// TwinCAT 3 PLC project Main
// ProgramVersion: 3.1.4024.0
// libraries:
//   Tc2_Standard, * (Beckhoff Automation GmbH)
//   Tc2_System, * (Beckhoff Automation GmbH)
//   Tc3_Module, * (Beckhoff Automation GmbH)
//   VisuDialogs, * (System)
//   VisuSymbols,3.5.10.0,System
// project tree:
//   DUTs/ AI_config.TcDUT, ST_DigitalIn.TcDUT, ST_DigitalOut.TcDUT, TC_config.TcDUT
//   FunctionBlocks/ c_to_f.TcPOU, FB_AnalogIn.TcPOU, FB_AnalogOut.TcPOU, FB_DigitalIn.TcPOU, FB_DigitalOut.TcPOU, FB_IOManager.TcPOU, FB_TCIn.TcPOU
//   Functions/ Count_to_MeasureUnits.TcPOU, MeasureUnits_to_Count.TcPOU, MeasureUnit_to_EngUnits.TcPOU, EngUnits_to_MeasureUnit.TcPOU
//   / GlobalTextList.TcGTLO, PlcTask.TcTTO, Visualization Manager.TcVMO (not stored)
//   GVLs/ GVL.TcGVL, GVL_AnalogInputs.TcGVL, GVL_AnalogOutputs.TcGVL, GVL_Counts.TcGVL, GVL_DigitalIn.TcGVL, GVL_DigitalOut.TcGVL, GVL_Thermocouples.TcGVL, HMI.TcGVL
//   POUs/ MAIN.TcPOU
//   VISUs/ rs1.TcVIS, rs2.TcVIS, rs3.TcVIS
// real-time tasks:
//   TASK PlcTask: cycle T#10ms, priority 20, ADS port 350
// I/O:
//   DEVICE Device 1 (EtherCAT) (disabled), AmsNetId 192.168.10.40.2.1
//     Term 1 (EK1100) [EK1100 EtherCAT Coupler (2A E-Bus)] (disabled)
//       Term 3 (EL1512) [EL1512 2Ch. +/- Counter 24V, 1kHz]
//       Term 2 (EL1512) [EL1512 2Ch. +/- Counter 24V, 1kHz]
//       Term 5 (EL2008) [EL2008 8Ch. Dig. Output 24V, 0.5A]
//       Term 4 (EL2008) [EL2008 8Ch. Dig. Output 24V, 0.5A]
//       Term 6 (EL3058) [EL3058 8Ch. Ana. Input 4-20mA]
//       Term 7 (EL3314) [EL3314 4Ch. Ana. Input Thermocouple (TC)]
//       Term 8 (EK1122) [EK1122 2 port EtherCAT junction]
//       Term 9 (EK1122) [EK1122 2 port EtherCAT junction]
//       Term 10 (EK1122) [EK1122 2 port EtherCAT junction]
// variable links:
//   Main/Main Instance <-> Device 1 (EtherCAT)/Term 1 (EK1100)/Term 4 (EL2008)
//     PlcTask Outputs/GVL_DigitalOut.bDigitalOut[{9..16}] <-> Channel {1..8}/Output  (8 links)
//   Main/Main Instance <-> Device 1 (EtherCAT)/Term 1 (EK1100)/Term 5 (EL2008)
//     PlcTask Outputs/GVL_DigitalOut.bDigitalOut[{1..8}] <-> Channel {1..8}/Output  (8 links)
//   Main/Main Instance <-> Device 1 (EtherCAT)/Term 1 (EK1100)/Term 6 (EL3058)
//     PlcTask Inputs/GVL_AnalogInputs.hmi_config[{1..8}].iRawCount <-> AI Standard Channel {1..8}/Value  (8 links)
//   Main/Main Instance <-> Device 1 (EtherCAT)/Term 1 (EK1100)/Term 7 (EL3314)
//     PlcTask Inputs/GVL_Thermocouples.hmi_config[{1..4}].iRawCountIn <-> TC Inputs Channel {1..4}/Value  (4 links)

CONFIGURATION Main
    RESOURCE PLC ON TwinCAT3
        TASK PlcTask(INTERVAL := T#10ms, PRIORITY := 20);
        PROGRAM MAIN WITH PlcTask : MAIN;
    END_RESOURCE
END_CONFIGURATION

// ---- DUTs/AI_config.TcDUT
TYPE AI_config :
STRUCT
	//{attribute 'OPC.UA.DA' := '1'}
	slope 				: REAL;
	//{attribute 'OPC.UA.DA' := '1'}
	offset 				: REAL;
	iRawCount AT %I*	: INT;
	rRawUnits			: REAL;
	//{attribute 'OPC.UA.DA' := '1'}
	rEngUnit 			: REAL;
	bDataValid 			: BOOL;
END_STRUCT
END_TYPE

// ---- DUTs/ST_DigitalIn.TcDUT
TYPE ST_DigitalIn :
STRUCT
	din 		: BOOL;
END_STRUCT
END_TYPE

// ---- DUTs/ST_DigitalOut.TcDUT
TYPE ST_DigitalOut :
STRUCT
	dout 		: BOOL;
	dout_fdbk			: BOOL;
END_STRUCT
END_TYPE

// ---- DUTs/TC_config.TcDUT
TYPE TC_config :
STRUCT
	iRawCountIn	AT %I*	: INT; 
	rTempC				: REAL;
	rTempF				: REAL;
END_STRUCT
END_TYPE

// ---- GVLs/GVL.TcGVL
VAR_GLOBAL CONSTANT
	MAX_CSV_ROWS 			: DINT := 1000000;
	MAX_CSV_COLUMNS 		: INT := 100;
	MAX_CSV_FIELD_LENGTH	: INT := 100;
	cMaxCSVFieldValueSize : INT := 0;
	//IMax_DigitalOut					: INT :=8;
END_VAR

// ---- GVLs/GVL_AnalogInputs.TcGVL
{attribute 'qualified_only'}
VAR_GLOBAL CONSTANT
	iAIChannelCount : INT := 50;
	
END_VAR
VAR_GLOBAL
	iAinChannel						: ARRAY [1..iAIChannelCount] OF INT;
END_VAR
VAR_GLOBAL PERSISTENT
	hmi_config 						: ARRAY [1..iAIChannelCount] OF AI_config ;
END_VAR

// ---- GVLs/GVL_AnalogOutputs.TcGVL
{attribute 'qualified_only'}
VAR_GLOBAL CONSTANT
	iAOChannelCount : INT := 50;
	
END_VAR
VAR_GLOBAL
	in_cmd								: ARRAY [1..iAOChannelCount] OF REAL;
	fdbk								: ARRAY [1..iAOChannelCount] OF REAL;
	iAO							AT %Q*	: ARRAY [1..iAOChannelCount] OF INT;
	ifdbk							AT %I*	: ARRAY [1..iAOChannelCount] OF INT;
END_VAR

// ---- GVLs/GVL_Counts.TcGVL
{attribute 'qualified_only'}
VAR_GLOBAL
	iCounter AT %I* : array[1..4] of UDINT;
END_VAR

// ---- GVLs/GVL_DigitalIn.TcGVL
{attribute 'qualified_only'}
VAR_GLOBAL CONSTANT
	iDinChannelCount : INT := 50;
END_VAR
VAR_GLOBAL
	bDigitalIn AT %I* : ARRAY [1..iDinChannelCount] OF BOOL;
	iDinChannel	: ARRAY [1..iDinChannelCount] OF INT;
	iEnabledChannels	: INT := 4;
END_VAR

// ---- GVLs/GVL_DigitalOut.TcGVL

VAR_GLOBAL CONSTANT
	iDoutputChannelCount : INT := 48;
END_VAR
VAR_GLOBAL
	bDigitalOut AT %Q*	: ARRAY [1..iDoutputChannelCount] OF BOOL;
	bDigitalOutFdbk : ARRAY [1..iDoutputChannelCount] OF BOOL;
	iDoutChannel	: ARRAY [1..iDoutputChannelCount] OF INT;
END_VAR

// ---- GVLs/GVL_Thermocouples.TcGVL
{attribute 'qualified_only'}
VAR_GLOBAL CONSTANT
	iTCchannelCount : INT := 20;
END_VAR
VAR_GLOBAL
	hmi_config 						: ARRAY [1..iTCchannelCount] OF TC_config ;
	iTCChannel						: ARRAY [1..20] OF INT;
END_VAR

// ---- GVLs/HMI.TcGVL
{attribute 'qualified_only'}
VAR_GLOBAL 
	
	bDigitalOcmd				: ARRAY[1..iDoutputChannelCount]OF BOOL;

END_VAR
VAR_GLOBAL PERSISTENT
	iEnabledChannels_DO,
	iEnabledChannels_DI,
	iEnabledChannels_AO,
	iEnabledChannels_AI,
	iEnabledChannels_TC			: INT;
END_VAR

// ---- POUs/MAIN.TcPOU
PROGRAM MAIN
VAR
	fbIO	: FB_IOManager;
END_VAR

fbIO();

END_PROGRAM

// ---- FunctionBlocks/FB_IOManager.TcPOU
FUNCTION_BLOCK FB_IOManager
VAR_INPUT
END_VAR
VAR_OUTPUT
END_VAR
VAR
	fbAI 	:	FB_Analogin;
	fbAO	:	FB_AnalogOut;
	fbDI	:	FB_DigitalIn;
	fbDO	:	FB_DigitalOut;
	fbTC	:	FB_TCIn;
END_VAR

(*
fbAI(iMaxInCH	:=	HMI.iEnabledChannels_AI);
fbAO(iMaxInCH	:=	HMI.iEnabledChannels_AO);
fbDI(iMaxInCH	:=	HMI.iEnabledChannels_DI);
fbDO(iMaxInCH	:=	HMI.iEnabledChannels_DO);
fbTC(iMaxInCH	:=	HMI.iEnabledChannels_TC);
*)

fbAI(iMaxInCH	:=	6);
fbAO(iMaxInCH	:=	3);
fbDI(iMaxInCH	:=	30);
fbDO(iMaxInCH	:=	16);
fbTC(iMaxInCH	:=	12);

END_FUNCTION_BLOCK

// ---- FunctionBlocks/FB_AnalogIn.TcPOU
FUNCTION_BLOCK FB_AnalogIn
VAR_INPUT 
	iMaxInCH : INT;
END_VAR
VAR_OUTPUT
END_VAR
VAR
	//AnalogIn	: ARRAY [1..GVL_AnalogInputs.iAIChannelCount] OF AI_config;
	iIndex 		: INT;
	iMax		: INT;
END_VAR

IF iMaxInCH > GVL_AnalogInputs.iAIChannelCount THEN
	iMax := GVL_AnalogInputs.iAIChannelCount;
ELSE
	iMax := iMaxInCH;
END_IF

FOR iIndex :=1 TO iMax BY 1 DO
	(*IF GVL_AnalogInputs.iAinChannel[iIndex]>0 THEN*)
	GVL_AnalogInputs.hmi_config[iIndex].rRawUnits:= Count_to_MeasureUnits
		(
		iValue_in	:=	GVL_AnalogInputs.hmi_config[iIndex].iRawCount,
		iHigh		:=	20,
		iLow		:= 	4
		);
		
	GVL_AnalogInputs.hmi_config[iIndex].rEngUnit:= MeasureUnit_to_EngUnits
		(	
		rValue:= GVL_AnalogInputs.hmi_config[iIndex].rRawUnits,
		rSlope:= GVL_AnalogInputs.hmi_config[iIndex].slope,
		rOffset:=GVL_AnalogInputs.hmi_config[iIndex].offset
		);
		
END_FOR

END_FUNCTION_BLOCK

// ---- Functions/Count_to_MeasureUnits.TcPOU
FUNCTION Count_to_MeasureUnits : REAL
VAR_INPUT
	iValue_in	: INT; 
	iHigh		: REAL;
	iLow		: REAL;
END_VAR
VAR
END_VAR

Count_to_MeasureUnits := ((iHigh - iLow) / 32767.0) * INT_TO_REAL(iValue_In) + iLow;

END_FUNCTION

// ---- Functions/MeasureUnit_to_EngUnits.TcPOU
FUNCTION MeasureUnit_to_EngUnits : REAL
VAR_INPUT
	rValue		: REAL;
	rSlope 		: REAL;
	rOffset 	: REAL;
END_VAR
VAR
END_VAR

MeasureUnit_to_EngUnits := (rValue*rSlope)+rOffset;

END_FUNCTION

// ---- FunctionBlocks/FB_AnalogOut.TcPOU
FUNCTION_BLOCK FB_AnalogOut
VAR_INPUT 
	iMaxInCH : INT;
END_VAR
VAR_OUTPUT
END_VAR
VAR
	//AnalogIn	: ARRAY [1..GVL_AnalogInputs.iAIChannelCount] OF AI_config;
	iIndex 		: INT;
	iMax		: INT;
END_VAR

IF iMaxInCH > GVL_AnalogOutputs.iAOChannelCount THEN
	iMax := GVL_AnalogOutputs.iAOChannelCount;
ELSE
	iMax := iMaxInCH;
END_IF

FOR iIndex :=1 TO iMax BY 1 DO
	//IF GVL_AnalogOutputs.in_cmd[iIndex] <= 4 or GVL_AnalogOutputs.in_cmd[iIndex]>20 THEN		// for 4-20mA
	IF GVL_AnalogOutputs.in_cmd[iIndex] <= 0 OR GVL_AnalogOutputs.in_cmd[iIndex]>100 THEN		// for percentage
		GVL_AnalogOutputs.iAO[iIndex]	:= 0;
	ELSE
		GVL_AnalogOutputs.iAO[iIndex]	:=	MeasureUnits_to_Count(iValue_in	:=	GVL_AnalogOutputs.in_cmd[iIndex],	iHigh:= 100,	iLow:=0);
		GVL_AnalogOutputs.fdbk[iIndex]	:=  Count_to_MeasureUnits(iValue_in :=  GVL_AnalogOutputs.ifdbk[iIndex],		iHigh:= 100,  	iLow:=0);
	END_IF
		
END_FOR

END_FUNCTION_BLOCK

// ---- Functions/MeasureUnits_to_Count.TcPOU
FUNCTION MeasureUnits_to_Count : int;
VAR_INPUT
	iValue_in	: REAL; 
	iHigh		: REAL;
	iLow		: REAL;
END_VAR
VAR
END_VAR

MeasureUnits_to_Count	:=	TO_INT(((iValue_In) - iLow)*(32767.0/(iHigh - iLow)));

END_FUNCTION

// ---- FunctionBlocks/FB_DigitalIn.TcPOU
FUNCTION_BLOCK FB_DigitalIn
VAR_INPUT
	iMaxInCH : INT;
END_VAR
VAR_OUTPUT
END_VAR
VAR
	arDinput 	: ARRAY [1..GVL_DigitalIn.iDinChannelCount] OF ST_DigitalIn;
	iIndex		: INT;
	iMax		: INT;
END_VAR

IF iMaxInCH > GVL_DigitalIn.iDinChannelCount THEN
	iMax := GVL_DigitalIn.iDinChannelCount;
ELSE
	iMax := iMaxInCH;
END_IF

FOR iIndex :=1 TO iMax BY 1 DO
	IF GVL_DigitalIn.iDinChannel[iIndex] > 0 THEN
		GVL_DigitalIn.bDigitalIn[GVL_DigitalIn.iDinChannel[iIndex]]:= arDinput[GVL_DigitalIn.iDinChannel[iIndex]].din;
	END_IF
END_FOR

END_FUNCTION_BLOCK

// ---- FunctionBlocks/FB_DigitalOut.TcPOU
FUNCTION_BLOCK FB_DigitalOut
VAR_INPUT
	iMaxInCH : INT;
END_VAR
VAR_OUTPUT
END_VAR
VAR

	arDigitalOut 	: ARRAY [1..GVL_DigitalOut.iDoutputChannelCount] OF ST_DigitalOut;
	bLocalDO		: ARRAY [1..GVL_DigitalOut.iDoutputChannelCount] OF BOOL;
	iIndex			: INT;
	iSeqIndex		: INT;
	iMax			: INT;
	arrtrig_output	: ARRAY [1..GVL_DigitalOut.iDoutputChannelCount] OF R_TRIG;
END_VAR
VAR PERSISTENT
	bSafetyDO		: ARRAY [1..GVL_DigitalOut.iDoutputChannelCount] OF BOOL;
END_VAR

AssignDOs();

METHOD AssignDOs : BOOL
VAR_INPUT
END_VAR
VAR
END_VAR
FOR iIndex:=1 TO iMaxInCH BY 1 DO
	GVL_DigitalOut.bDigitalOutFdbk[iIndex] := OutputControl;
END_FOR
END_METHOD

METHOD AssignSafetyChannels : BOOL
VAR_INPUT
END_VAR
bSafetyDO[1]:=TRUE;
bSafetyDO[2]:=TRUE;
bSafetyDO[3]:=TRUE;
bSafetyDO[4]:=TRUE;
END_METHOD

METHOD LimitMaxChannels : BOOL
(*IF iMaxInCH > GVL_DigitalOut.iDoutputChannelCount THEN
	iMax := GVL_DigitalOut.iDoutputChannelCount;
ELSE
	iMax := iMaxInCH;
END_IF
*)

iMax := GVL_DigitalOut.iDoutputChannelCount;
END_METHOD

PROPERTY OutputControl : BOOL
GET
OutputControl:=GVL_DigitalOut.bDigitalOut[iIndex];
END_GET
SET
GVL_DigitalOut.bDigitalOut[iIndex] := OutputControl;
END_SET
END_PROPERTY

END_FUNCTION_BLOCK

// ---- FunctionBlocks/FB_TCIn.TcPOU
FUNCTION_BLOCK FB_TCIn
VAR_INPUT
	iMaxInCH : INT;
END_VAR
VAR_OUTPUT
END_VAR
VAR
	iIndex 		: INT;
	iMax		: INT;
END_VAR

IF iMaxInCH > GVL_Thermocouples.iTCchannelCount THEN
	iMax := GVL_Thermocouples.iTCchannelCount;
ELSE
	iMax := iMaxInCH;
END_IF

FOR iIndex :=1 TO iMax BY 1 DO 

	GVL_Thermocouples.hmi_config[iIndex].rTempC	:= TO_REAL(GVL_Thermocouples.hmi_config[iIndex].iRawCountIn)/10;
	GVL_Thermocouples.hmi_config[iIndex].rTempF	:=c_to_f
		(
		tempC:=GVL_Thermocouples.hmi_config[iIndex].rTempC
		);
END_FOR

END_FUNCTION_BLOCK

// ---- FunctionBlocks/c_to_f.TcPOU
FUNCTION c_to_f : REAL
VAR_INPUT
	tempC : REAL;
END_VAR
VAR
END_VAR

c_to_f := (tempC*1.8) + 32;

END_FUNCTION

// ---- Functions/EngUnits_to_MeasureUnit.TcPOU
FUNCTION EngUnits_to_MeasureUnit : REAL
VAR_INPUT
	rValue		: REAL;
	rSlope 		: REAL;
	rOffset 	: REAL;
END_VAR
VAR
END_VAR

MeasureUnit_to_EngUnits := (rValue*rSlope)+rOffset;

END_FUNCTION

// ---- GlobalTextList.TcGTLO
TEXTLIST GlobalTextList
  592 = '%'
  352 = '%s'
  613 = 'AI#'
  186 = 'AI1'
  998 = 'AI1 (PT01)'
  490 = 'AI2'
  67 = 'AI2 (PT01)'
  824 = 'AI3'
  817 = 'AI4'
  563 = 'AMSNetID'
  293 = 'AO#'
  746 = 'AO1'
  550 = 'AO1  (PCV01)'
  84 = 'AO1 -(PCV01)'
  87 = 'AO2'
  522 = 'AO3'
  463 = 'AO4'
  764 = 'bar'
  586 = 'CH1'
  207 = 'CH2'
  901 = 'CH3'
  498 = 'CH4'
  972 = 'CH5'
  370 = 'CH6'
  416 = 'CH7'
  736 = 'CH8'
  868 = 'Channel 0/1'
  793 = 'Channel 1'
  734 = 'Channel 1 (XV02)'
  806 = 'Channel 1/2'
  108 = 'Channel 10 (XV05)'
  758 = 'Channel 10/12'
  59 = 'Channel 11 (XV05)'
  410 = 'Channel 12 (XV06)'
  615 = 'Channel 13 (XV02)'
  591 = 'Channel 13 (XV06)'
  268 = 'Channel 14 (XV02)'
  645 = 'Channel 14 (XV07)'
  555 = 'Channel 15 (XV07)'
  735 = 'Channel 2'
  895 = 'Channel 2 (XV04)'
  483 = 'Channel 2/3'
  760 = 'Channel 3'
  193 = 'Channel 3 (XV05)'
  6 = 'Channel 3/4'
  250 = 'Channel 4'
  105 = 'Channel 4 (XV06)'
  237 = 'Channel 4/5'
  314 = 'Channel 5'
  260 = 'Channel 5 (XV07)'
  408 = 'Channel 5/6'
  660 = 'Channel 6'
  80 = 'Channel 6/7'
  792 = 'Channel 7'
  318 = 'Channel 7/8'
  493 = 'Channel 8'
  918 = 'Channel 8 (XV04)'
  53 = 'Channel 9'
  523 = 'Channel 9 (XV04)'
  643 = 'Channel 9/10'
  479 = 'Channel 9/11'
  177 = 'Close'
  533 = 'Control'
  957 = 'Counter1'
  774 = 'Counter2'
  273 = 'Counter3'
  499 = 'Counter4'
  437 = 'DI#'
  129 = 'DigitalInputs'
  402 = 'DO#'
  407 = 'Feedback'
  859 = 'FilePath'
  350 = 'Manual Record'
  628 = 'Mxx-x100-TT06'
  281 = 'Mxx-x200-TT06'
  146 = 'Mxx-x300-TT06'
  209 = 'Mxx-x400-TT06'
  747 = 'Offset'
  816 = 'Open'
  394 = 'Output Button'
  928 = 'PCV01'
  270 = 'PT01'
  528 = 'Recording Rate'
  848 = 'Sequence Start'
  652 = 'Slope'
  280 = 'SoftwareStop'
  427 = 'TC#'
  572 = 'TC1 (Mxx-x100-TT06)'
  86 = 'TC2 (Mxx-x200-TT06)'
  707 = 'TC3 (Mxx-x300-TT06)'
  266 = 'TC4 (Mxx-x400-TT06)'
  549 = 'ToggleRate'
  360 = '°C'
END_TEXTLIST

// ---- VISUs/rs1.TcVIS
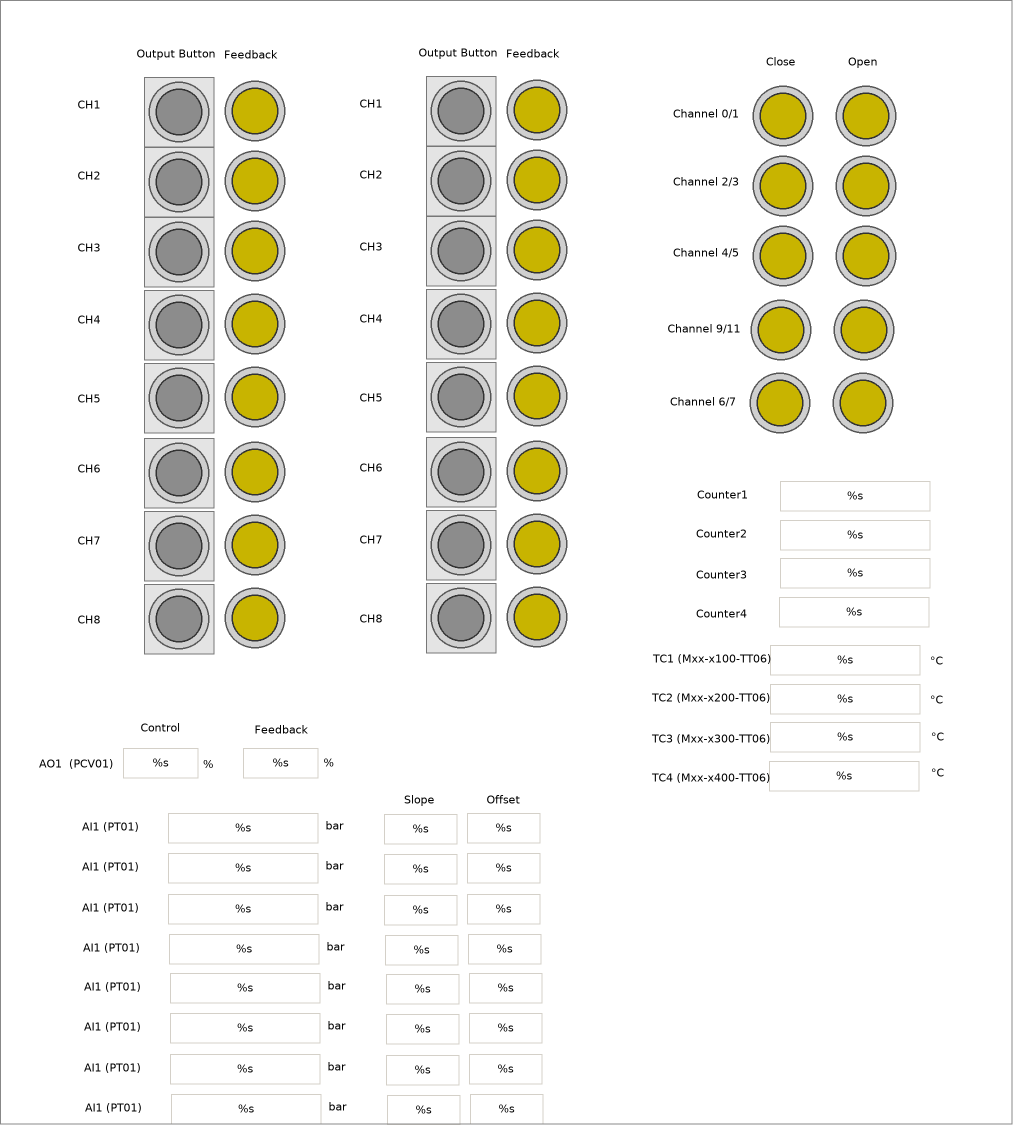
VISUALIZATION rs1  // 1013x1125
    Lamp1 (220,289 70x70), variable: bDigitalOutFdbk[4], style: Lamp-Lamp1-Yellow
    PushSwitch (144,290 70x70), variable: bDigitalOut[4], behaviour: TOGGLE, style: Switch-PushSwitch-Gray
    PushSwitch (144,77 70x70), variable: bDigitalOut[1], behaviour: TOGGLE, style: Switch-PushSwitch-Gray
    PushSwitch (144,147 70x70), variable: bDigitalOut[2], behaviour: TOGGLE, style: Switch-PushSwitch-Gray
    PushSwitch (144,217 70x70), variable: bDigitalOut[3], behaviour: TOGGLE, style: Switch-PushSwitch-Gray
    PushSwitch (144,363 70x70), variable: bDigitalOut[5], behaviour: TOGGLE, style: Switch-PushSwitch-Gray
    Lamp1 (220,76 70x70), variable: bDigitalOutFdbk[1], style: Lamp-Lamp1-Yellow
    Lamp1 (220,146 70x70), variable: bDigitalOutFdbk[2], style: Lamp-Lamp1-Yellow
    Lamp1 (220,216 70x70), variable: bDigitalOutFdbk[3], style: Lamp-Lamp1-Yellow
    Lamp1 (220,362 70x70), variable: bDigitalOutFdbk[5], style: Lamp-Lamp1-Yellow
    Label (101,39 150x30), "Output Button"
    Label (176,40 150x30), "Feedback"
    Label (14,305 150x30), "CH4"
    Label (14,90 150x30), "CH1"
    Label (14,161 150x30), "CH2"
    Label (14,233 150x30), "CH3"
    Label (14,384 150x30), "CH5"
    Lamp1 (748,81 70x70), variable: GVL_DigitalIn.bDigitalIn[1], style: Lamp-Lamp1-Yellow
    Lamp1 (831,81 70x70), variable: GVL_DigitalIn.bDigitalIn[2], style: Lamp-Lamp1-Yellow
    Lamp1 (748,151 70x70), variable: GVL_DigitalIn.bDigitalIn[3], style: Lamp-Lamp1-Yellow
    Lamp1 (831,151 70x70), variable: GVL_DigitalIn.bDigitalIn[4], style: Lamp-Lamp1-Yellow
    Lamp1 (748,221 70x70), variable: GVL_DigitalIn.bDigitalIn[5], style: Lamp-Lamp1-Yellow
    Lamp1 (831,221 70x70), variable: GVL_DigitalIn.bDigitalIn[6], style: Lamp-Lamp1-Yellow
    Lamp1 (745,368 70x70), variable: GVL_DigitalIn.bDigitalIn[7], style: Lamp-Lamp1-Yellow
    Lamp1 (828,368 70x70), variable: GVL_DigitalIn.bDigitalIn[8], style: Lamp-Lamp1-Yellow
    Label (631,99 150x30), "Channel 0/1"
    Label (631,167 150x30), "Channel 2/3"
    Label (631,238 150x30), "Channel 4/5"
    Label (628,387 150x30), "Channel 6/7"
    Textfield (770,645 150x30), "%s", text variable: GVL_Thermocouples.hmi_config[1].rTempC
    Label (637,644 151x30), "TC1 (Mxx-x100-TT06)"
    Textfield (770,684 150x30), "%s", text variable: GVL_Thermocouples.hmi_config[2].rTempC
    Textfield (770,722 150x30), "%s", text variable: GVL_Thermocouples.hmi_config[3].rTempC
    Textfield (769,761 150x30), "%s", text variable: GVL_Thermocouples.hmi_config[4].rTempC
    Label (706,47 150x30), "Close"
    Label (788,47 150x30), "Open"
    Label (636,683 151x30), "TC2 (Mxx-x200-TT06)"
    Label (636,724 151x30), "TC3 (Mxx-x300-TT06)"
    Label (636,763 151x30), "TC4 (Mxx-x400-TT06)"
    Textfield (123,748 75x30), "%s", text variable: GVL_AnalogOutputs.in_cmd[1]
        OnMouseDown: write the text variable via Default
    Label (1,749 151x30), "AO1 (PCV01)"
    Label (193,749 31x31), "%"
    Textfield (243,748 75x30), "%s", text variable: GVL_AnalogOutputs.fdbk[1]
    Label (314,748 30x30), "%"
    Label (206,715 151x30), "Feedback"
    Label (85,713 151x30), "Control"
    Label (861,646 151x30), "°C"
    Label (861,685 151x30), "°C"
    Label (862,722 151x30), "°C"
    Label (862,758 151x30), "°C"
    Textfield (168,813 150x30), "%s", text variable: GVL_AnalogInputs.hmi_config[1].rEngUnit
    Label (35,812 151x30), "AI1 (PT01)"
    Label (311,811 47x30), "bar"
    Textfield (384,814 73x30), "%s", text variable: GVL_AnalogInputs.hmi_config[1].slope
        OnMouseDown: write the text variable via Default
    Textfield (467,813 73x30), "%s", text variable: GVL_AnalogInputs.hmi_config[1].offset
        OnMouseDown: write the text variable via Default
    Label (382,785 75x30), "Slope"
    Label (466,785 75x30), "Offset"
    Lamp1 (746,295 70x70), variable: GVL_DigitalIn.bDigitalIn[9], style: Lamp-Lamp1-Yellow
    Lamp1 (829,295 70x70), variable: GVL_DigitalIn.bDigitalIn[10], style: Lamp-Lamp1-Yellow
    Label (629,314 150x30), "Channel 9/11"
    Lamp1 (220,510 70x70), variable: bDigitalOutFdbk[7], style: Lamp-Lamp1-Yellow
    PushSwitch (144,511 70x70), variable: bDigitalOut[7], behaviour: TOGGLE, style: Switch-PushSwitch-Gray
    PushSwitch (144,438 70x70), variable: bDigitalOut[6], behaviour: TOGGLE, style: Switch-PushSwitch-Gray
    PushSwitch (144,584 70x70), variable: bDigitalOut[8], behaviour: TOGGLE, style: Switch-PushSwitch-Gray
    Lamp1 (220,437 70x70), variable: bDigitalOutFdbk[6], style: Lamp-Lamp1-Yellow
    Lamp1 (220,583 70x70), variable: bDigitalOutFdbk[8], style: Lamp-Lamp1-Yellow
    Label (14,526 150x30), "CH7"
    Label (14,454 150x30), "CH6"
    Label (14,605 150x30), "CH8"
    Lamp1 (502,288 70x70), variable: bDigitalOutFdbk[12], style: Lamp-Lamp1-Yellow
    PushSwitch (426,289 70x70), variable: bDigitalOut[12], behaviour: TOGGLE, style: Switch-PushSwitch-Gray
    PushSwitch (426,76 70x70), variable: bDigitalOut[9], behaviour: TOGGLE, style: Switch-PushSwitch-Gray
    PushSwitch (426,146 70x70), variable: bDigitalOut[10], behaviour: TOGGLE, style: Switch-PushSwitch-Gray
    PushSwitch (426,216 70x70), variable: bDigitalOut[11], behaviour: TOGGLE, style: Switch-PushSwitch-Gray
    PushSwitch (426,362 70x70), variable: bDigitalOut[13], behaviour: TOGGLE, style: Switch-PushSwitch-Gray
    Lamp1 (502,75 70x70), variable: bDigitalOutFdbk[9], style: Lamp-Lamp1-Yellow
    Lamp1 (502,145 70x70), variable: bDigitalOutFdbk[10], style: Lamp-Lamp1-Yellow
    Lamp1 (502,215 70x70), variable: bDigitalOutFdbk[11], style: Lamp-Lamp1-Yellow
    Lamp1 (502,361 70x70), variable: bDigitalOutFdbk[13], style: Lamp-Lamp1-Yellow
    Label (383,38 150x30), "Output Button"
    Label (458,39 150x30), "Feedback"
    Label (296,304 150x30), "CH4"
    Label (296,89 150x30), "CH1"
    Label (296,160 150x30), "CH2"
    Label (296,232 150x30), "CH3"
    Label (296,383 150x30), "CH5"
    Lamp1 (502,509 70x70), variable: bDigitalOutFdbk[15], style: Lamp-Lamp1-Yellow
    PushSwitch (426,510 70x70), variable: bDigitalOut[15], behaviour: TOGGLE, style: Switch-PushSwitch-Gray
    PushSwitch (426,437 70x70), variable: bDigitalOut[14], behaviour: TOGGLE, style: Switch-PushSwitch-Gray
    PushSwitch (426,583 70x70), variable: bDigitalOut[16], behaviour: TOGGLE, style: Switch-PushSwitch-Gray
    Lamp1 (502,436 70x70), variable: bDigitalOutFdbk[14], style: Lamp-Lamp1-Yellow
    Lamp1 (502,582 70x70), variable: bDigitalOutFdbk[16], style: Lamp-Lamp1-Yellow
    Label (296,525 150x30), "CH7"
    Label (296,453 150x30), "CH6"
    Label (296,604 150x30), "CH8"
    Textfield (780,481 150x30), "%s", text variable: GVL_Counts.iCounter[1]
    Label (647,480 151x30), "Counter1"
    Textfield (780,520 150x30), "%s", text variable: GVL_Counts.iCounter[2]
    Textfield (780,558 150x30), "%s", text variable: GVL_Counts.iCounter[3]
    Textfield (779,597 150x30), "%s", text variable: GVL_Counts.iCounter[4]
    Label (646,519 151x30), "Counter2"
    Label (646,560 151x30), "Counter3"
    Label (646,599 151x30), "Counter4"
    Textfield (168,853 150x30), "%s", text variable: GVL_AnalogInputs.hmi_config[1].rEngUnit
    Label (35,852 151x30), "AI1 (PT01)"
    Label (311,851 47x30), "bar"
    Textfield (384,854 73x30), "%s", text variable: GVL_AnalogInputs.hmi_config[2].slope
        OnMouseDown: write the text variable via Default
    Textfield (467,853 73x30), "%s", text variable: GVL_AnalogInputs.hmi_config[2].offset
        OnMouseDown: write the text variable via Default
    Textfield (168,894 150x30), "%s", text variable: GVL_AnalogInputs.hmi_config[3].rEngUnit
    Label (35,893 151x30), "AI1 (PT01)"
    Label (311,892 47x30), "bar"
    Textfield (384,895 73x30), "%s", text variable: GVL_AnalogInputs.hmi_config[3].slope
        OnMouseDown: write the text variable via Default
    Textfield (467,894 73x30), "%s", text variable: GVL_AnalogInputs.hmi_config[3].offset
        OnMouseDown: write the text variable via Default
    Textfield (169,934 150x30), "%s", text variable: GVL_AnalogInputs.hmi_config[4].rEngUnit
    Label (36,933 151x30), "AI1 (PT01)"
    Label (312,932 47x30), "bar"
    Textfield (385,935 73x30), "%s", text variable: GVL_AnalogInputs.hmi_config[4].slope
        OnMouseDown: write the text variable via Default
    Textfield (468,934 73x30), "%s", text variable: GVL_AnalogInputs.hmi_config[4].offset
        OnMouseDown: write the text variable via Default
    Textfield (170,973 150x30), "%s", text variable: GVL_AnalogInputs.hmi_config[5].rEngUnit
    Label (37,972 151x30), "AI1 (PT01)"
    Label (313,971 47x30), "bar"
    Textfield (386,974 73x30), "%s", text variable: GVL_AnalogInputs.hmi_config[5].slope
        OnMouseDown: write the text variable via Default
    Textfield (469,973 73x30), "%s", text variable: GVL_AnalogInputs.hmi_config[5].offset
        OnMouseDown: write the text variable via Default
    Textfield (170,1013 150x30), "%s", text variable: GVL_AnalogInputs.hmi_config[6].rEngUnit
    Label (37,1012 151x30), "AI1 (PT01)"
    Label (313,1011 47x30), "bar"
    Textfield (386,1014 73x30), "%s", text variable: GVL_AnalogInputs.hmi_config[6].slope
        OnMouseDown: write the text variable via Default
    Textfield (469,1013 73x30), "%s", text variable: GVL_AnalogInputs.hmi_config[6].offset
        OnMouseDown: write the text variable via Default
    Textfield (170,1054 150x30), "%s", text variable: GVL_AnalogInputs.hmi_config[7].rEngUnit
    Label (37,1053 151x30), "AI1 (PT01)"
    Label (313,1052 47x30), "bar"
    Textfield (386,1055 73x30), "%s", text variable: GVL_AnalogInputs.hmi_config[7].slope
        OnMouseDown: write the text variable via Default
    Textfield (469,1054 73x30), "%s", text variable: GVL_AnalogInputs.hmi_config[7].offset
        OnMouseDown: write the text variable via Default
    Textfield (171,1094 150x30), "%s", text variable: GVL_AnalogInputs.hmi_config[8].rEngUnit
    Label (38,1093 151x30), "AI1 (PT01)"
    Label (314,1092 47x30), "bar"
    Textfield (387,1095 73x30), "%s", text variable: GVL_AnalogInputs.hmi_config[8].slope
        OnMouseDown: write the text variable via Default
    Textfield (470,1094 73x30), "%s", text variable: GVL_AnalogInputs.hmi_config[8].offset
        OnMouseDown: write the text variable via Default
END_VISUALIZATION

// ---- VISUs/rs2.TcVIS
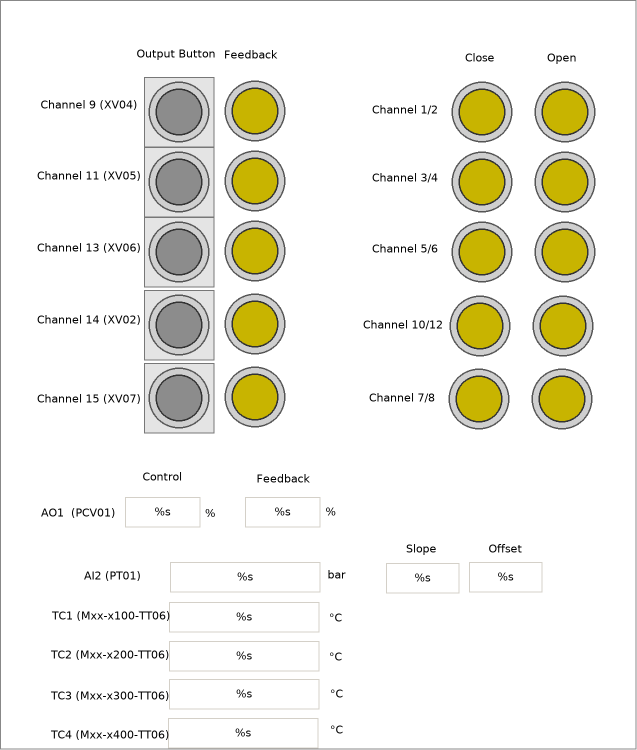
VISUALIZATION rs2  // 637x750
    Lamp1 (220,289 70x70), variable: bDigitalOutFdbk[9], style: Lamp-Lamp1-Yellow
    PushSwitch (144,290 70x70), variable: bDigitalOut[9], behaviour: TOGGLE, style: Switch-PushSwitch-Gray
    PushSwitch (144,77 70x70), variable: bDigitalOut[6], behaviour: TOGGLE, style: Switch-PushSwitch-Gray
    PushSwitch (144,147 70x70), variable: bDigitalOut[7], behaviour: TOGGLE, style: Switch-PushSwitch-Gray
    PushSwitch (144,217 70x70), variable: bDigitalOut[8], behaviour: TOGGLE, style: Switch-PushSwitch-Gray
    PushSwitch (144,363 70x70), variable: bDigitalOut[10], behaviour: TOGGLE, style: Switch-PushSwitch-Gray
    Lamp1 (220,76 70x70), variable: bDigitalOutFdbk[6], style: Lamp-Lamp1-Yellow
    Lamp1 (220,146 70x70), variable: bDigitalOutFdbk[7], style: Lamp-Lamp1-Yellow
    Lamp1 (220,216 70x70), variable: bDigitalOutFdbk[8], style: Lamp-Lamp1-Yellow
    Lamp1 (220,362 70x70), variable: bDigitalOutFdbk[10], style: Lamp-Lamp1-Yellow
    Label (101,39 150x30), "Output Button"
    Label (176,40 150x30), "Feedback"
    Label (14,305 150x30), "Channel 14 (XV02)"
    Label (14,90 150x30), "Channel 9 (XV04)"
    Label (14,161 150x30), "Channel 11 (XV05)"
    Label (14,233 150x30), "Channel 13 (XV06)"
    Label (14,384 150x30), "Channel 15 (XV07)"
    Lamp1 (447,77 70x70), variable: GVL_DigitalIn.bDigitalIn[11], style: Lamp-Lamp1-Yellow
    Lamp1 (530,77 70x70), variable: GVL_DigitalIn.bDigitalIn[12], style: Lamp-Lamp1-Yellow
    Lamp1 (447,147 70x70), variable: GVL_DigitalIn.bDigitalIn[13], style: Lamp-Lamp1-Yellow
    Lamp1 (530,147 70x70), variable: GVL_DigitalIn.bDigitalIn[14], style: Lamp-Lamp1-Yellow
    Lamp1 (447,217 70x70), variable: GVL_DigitalIn.bDigitalIn[15], style: Lamp-Lamp1-Yellow
    Lamp1 (530,217 70x70), variable: GVL_DigitalIn.bDigitalIn[16], style: Lamp-Lamp1-Yellow
    Lamp1 (444,364 70x70), variable: GVL_DigitalIn.bDigitalIn[17], style: Lamp-Lamp1-Yellow
    Lamp1 (527,364 70x70), variable: GVL_DigitalIn.bDigitalIn[18], style: Lamp-Lamp1-Yellow
    Label (330,95 150x30), "Channel 1/2"
    Label (330,163 150x30), "Channel 3/4"
    Label (330,234 150x30), "Channel 5/6"
    Label (327,383 150x30), "Channel 7/8"
    Textfield (169,602 150x30), "%s", text variable: GVL_Thermocouples.hmi_config[5].rTempC
    Label (36,601 151x30), "TC1 (Mxx-x100-TT06)"
    Textfield (169,641 150x30), "%s", text variable: GVL_Thermocouples.hmi_config[6].rTempC
    Textfield (169,679 150x30), "%s", text variable: GVL_Thermocouples.hmi_config[7].rTempC
    Textfield (168,718 150x30), "%s", text variable: GVL_Thermocouples.hmi_config[8].rTempC
    Label (405,43 150x30), "Close"
    Label (487,43 150x30), "Open"
    Label (35,640 151x30), "TC2 (Mxx-x200-TT06)"
    Label (35,681 151x30), "TC3 (Mxx-x300-TT06)"
    Label (35,720 151x30), "TC4 (Mxx-x400-TT06)"
    Textfield (125,497 75x30), "%s", text variable: GVL_AnalogOutputs.in_cmd[2]
        OnMouseDown: write the text variable via Default
    Label (3,498 151x30), "AO1 (PCV01)"
    Label (195,498 31x31), "%"
    Textfield (245,497 75x30), "%s", text variable: GVL_AnalogOutputs.fdbk[2]
    Label (316,497 30x30), "%"
    Label (208,464 151x30), "Feedback"
    Label (87,462 151x30), "Control"
    Label (260,603 151x30), "°C"
    Label (260,642 151x30), "°C"
    Label (261,679 151x30), "°C"
    Label (261,715 151x30), "°C"
    Textfield (170,562 150x30), "%s", text variable: GVL_AnalogInputs.hmi_config[2].rEngUnit
    Label (37,561 151x30), "AI2 (PT01)"
    Label (313,560 47x30), "bar"
    Textfield (386,563 73x30), "%s", text variable: GVL_AnalogInputs.hmi_config[2].slope
        OnMouseDown: write the text variable via Default
    Textfield (469,562 73x30), "%s", text variable: GVL_AnalogInputs.hmi_config[2].offset
        OnMouseDown: write the text variable via Default
    Label (384,534 75x30), "Slope"
    Label (468,534 75x30), "Offset"
    Lamp1 (445,291 70x70), variable: GVL_DigitalIn.bDigitalIn[19], style: Lamp-Lamp1-Yellow
    Lamp1 (528,291 70x70), variable: GVL_DigitalIn.bDigitalIn[20], style: Lamp-Lamp1-Yellow
    Label (328,310 150x30), "Channel 10/12"
END_VISUALIZATION

// ---- VISUs/rs3.TcVIS
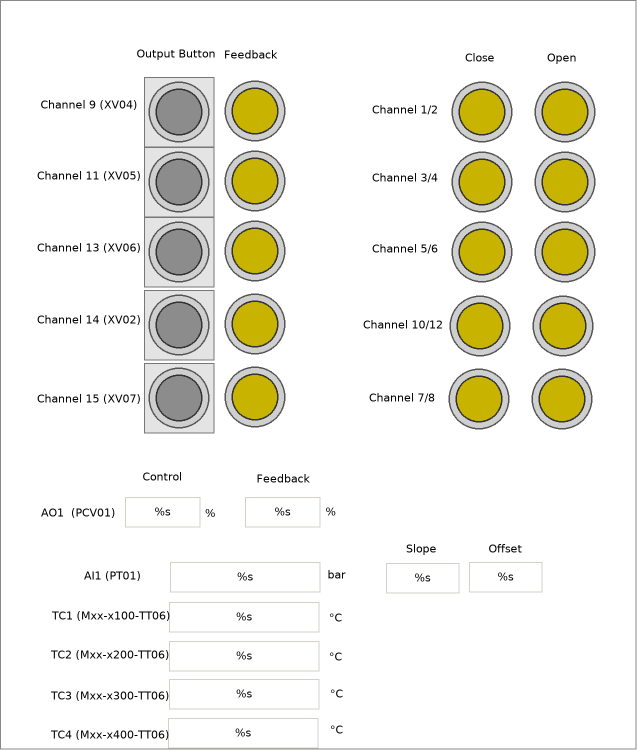
VISUALIZATION rs3  // 637x750
    Lamp1 (220,289 70x70), variable: bDigitalOutFdbk[14], style: Lamp-Lamp1-Yellow
    PushSwitch (144,290 70x70), variable: bDigitalOut[14], behaviour: TOGGLE, style: Switch-PushSwitch-Gray
    PushSwitch (144,77 70x70), variable: bDigitalOut[11], behaviour: TOGGLE, style: Switch-PushSwitch-Gray
    PushSwitch (144,147 70x70), variable: bDigitalOut[12], behaviour: TOGGLE, style: Switch-PushSwitch-Gray
    PushSwitch (144,217 70x70), variable: bDigitalOut[13], behaviour: TOGGLE, style: Switch-PushSwitch-Gray
    PushSwitch (144,363 70x70), variable: bDigitalOut[15], behaviour: TOGGLE, style: Switch-PushSwitch-Gray
    Lamp1 (220,76 70x70), variable: bDigitalOutFdbk[11], style: Lamp-Lamp1-Yellow
    Lamp1 (220,146 70x70), variable: bDigitalOutFdbk[12], style: Lamp-Lamp1-Yellow
    Lamp1 (220,216 70x70), variable: bDigitalOutFdbk[13], style: Lamp-Lamp1-Yellow
    Lamp1 (220,362 70x70), variable: bDigitalOutFdbk[15], style: Lamp-Lamp1-Yellow
    Label (101,39 150x30), "Output Button"
    Label (176,40 150x30), "Feedback"
    Label (14,305 150x30), "Channel 14 (XV02)"
    Label (14,90 150x30), "Channel 9 (XV04)"
    Label (14,161 150x30), "Channel 11 (XV05)"
    Label (14,233 150x30), "Channel 13 (XV06)"
    Label (14,384 150x30), "Channel 15 (XV07)"
    Lamp1 (447,77 70x70), variable: GVL_DigitalIn.bDigitalIn[21], style: Lamp-Lamp1-Yellow
    Lamp1 (530,77 70x70), variable: GVL_DigitalIn.bDigitalIn[22], style: Lamp-Lamp1-Yellow
    Lamp1 (447,147 70x70), variable: GVL_DigitalIn.bDigitalIn[23], style: Lamp-Lamp1-Yellow
    Lamp1 (530,147 70x70), variable: GVL_DigitalIn.bDigitalIn[24], style: Lamp-Lamp1-Yellow
    Lamp1 (447,217 70x70), variable: GVL_DigitalIn.bDigitalIn[25], style: Lamp-Lamp1-Yellow
    Lamp1 (530,217 70x70), variable: GVL_DigitalIn.bDigitalIn[26], style: Lamp-Lamp1-Yellow
    Lamp1 (444,364 70x70), variable: GVL_DigitalIn.bDigitalIn[27], style: Lamp-Lamp1-Yellow
    Lamp1 (527,364 70x70), variable: GVL_DigitalIn.bDigitalIn[28], style: Lamp-Lamp1-Yellow
    Label (330,95 150x30), "Channel 1/2"
    Label (330,163 150x30), "Channel 3/4"
    Label (330,234 150x30), "Channel 5/6"
    Label (327,383 150x30), "Channel 7/8"
    Textfield (169,602 150x30), "%s", text variable: GVL_Thermocouples.hmi_config[9].rTempC
    Label (36,601 151x30), "TC1 (Mxx-x100-TT06)"
    Textfield (169,641 150x30), "%s", text variable: GVL_Thermocouples.hmi_config[10].rTempC
    Textfield (169,679 150x30), "%s", text variable: GVL_Thermocouples.hmi_config[11].rTempC
    Textfield (168,718 150x30), "%s", text variable: GVL_Thermocouples.hmi_config[12].rTempC
    Label (405,43 150x30), "Close"
    Label (487,43 150x30), "Open"
    Label (35,640 151x30), "TC2 (Mxx-x200-TT06)"
    Label (35,681 151x30), "TC3 (Mxx-x300-TT06)"
    Label (35,720 151x30), "TC4 (Mxx-x400-TT06)"
    Textfield (125,497 75x30), "%s", text variable: GVL_AnalogOutputs.in_cmd[3]
        OnMouseDown: write the text variable via Default
    Label (3,498 151x30), "AO1 (PCV01)"
    Label (195,498 31x31), "%"
    Textfield (245,497 75x30), "%s", text variable: GVL_AnalogOutputs.fdbk[3]
    Label (316,497 30x30), "%"
    Label (208,464 151x30), "Feedback"
    Label (87,462 151x30), "Control"
    Label (260,603 151x30), "°C"
    Label (260,642 151x30), "°C"
    Label (261,679 151x30), "°C"
    Label (261,715 151x30), "°C"
    Textfield (170,562 150x30), "%s", text variable: GVL_AnalogInputs.hmi_config[3].rEngUnit
    Label (37,561 151x30), "AI1 (PT01)"
    Label (313,560 47x30), "bar"
    Textfield (386,563 73x30), "%s", text variable: GVL_AnalogInputs.hmi_config[3].slope
        OnMouseDown: write the text variable via Default
    Textfield (469,562 73x30), "%s", text variable: GVL_AnalogInputs.hmi_config[3].offset
        OnMouseDown: write the text variable via Default
    Label (384,534 75x30), "Slope"
    Label (468,534 75x30), "Offset"
    Lamp1 (445,291 70x70), variable: GVL_DigitalIn.bDigitalIn[29], style: Lamp-Lamp1-Yellow
    Lamp1 (528,291 70x70), variable: GVL_DigitalIn.bDigitalIn[30], style: Lamp-Lamp1-Yellow
    Label (328,310 150x30), "Channel 10/12"
END_VISUALIZATION
